PROGRAM MAIN
VAR
	myEnum : (MY_THIS,MY_THAT);
	myDutEnum : MY_DUT_ENUM;
END_VAR

END_PROGRAM

(* stored: Version 1.1.0.1, ProductVersion 3.1.4024.12
   POU MAIN: Id {4f7f124e-2b6e-4c71-87e2-245c0f9c49a6}, SpecialFunc None *)
